# EPICS substitutions: BEAMCORR/BEAMCORR-IOC-01App/Db/coefficients.substitutions
file coefficients.template {
    pattern { INT_MAG, INP, DIRECTION}
    { "HIFI", "A", "MAIN"}
    { "HIFI", "B", "TRANS_X" }
    { "HIFI", "C", "TRANS_Y"}
    { "EMU", "D", "MAIN"}
    { "EMU", "E", "TRANS" }
    { "MUSR", "F", "MAIN"}
    { "MUSR", "G" "TRANS" }
}
